# EPICS StreamDevice protocol: protocols/acq2106clk.proto
Terminator = LF;
ExtraInput = Ignore;

getSi5326config {
	out "si5326config";
	in "%s";
}

setSi5326config {
	out "load.si5326 si5326_33M333-%dM.txt";
	in;
}
getSi5326bypass {
	out "si5326bypass";
	in "%d";
}

setSi5326Bypass {
	out "set_si5326_bypass %d";
	in;
}

acq480_init_clk {
	out "acq480_init_clk %dM";
	in;
}
